(* Logix 5000 project; controller WWTP_SEC_CLX vendor 1 type 14 code 54 rev 17.2; software revision 17.00; part 11 of 13 *)

VAR_GLOBAL   (* controller tags *)
   BLR400_Fault : P_DIn := (Inp_Gate := 1, Cfg_NormTextVis := 1, Cfg_PCmdClear := 1, Cfg_HasTgtDisagreeAlm := 1, Cfg_TgtDisagreeAckReqd := 1, Cfg_TgtDisagreeSeverity := 3, Cfg_TgtDisagreeMinDuration := 5, Sts_SubstPV := 1, Ack_TgtDisagree := 1, Rdy_InpPV := 1);   // Secondary Treatment BLR-400 Fault
   BLR400_Intlk : P_Intlk := (Cfg_Latched := 2#0000_0000_0000_0001, Cfg_Bypassable := 2#0000_0000_0000_0001, Cfg_PCmdClear := 1, Sts_NBIntlkOK := 1, Sts_Intlk := 2#0000_0000_0000_0001, Sts_FirstOut := 2#0000_0000_0000_0001, Rdy_Reset := 1);   // BLR-400 Interlock
   BLR400_Motor : P_Motor := (Inp_PermOK := 1, Inp_NBPermOK := 1, Inp_NBIntlkOK := 1, Cfg_HasRunFdbk := 1, Cfg_UseRunFdbk := 1, Cfg_HasPermObj := 1, Cfg_HasIntlkObj := 1, Cfg_HasResInhObj := 1, Cfg_HasRunTimeObj := 1, Cfg_HasFailToStartAlm := 1, Cfg_HasFailToStopAlm := 1, Cfg_HasIntlkTripAlm := 1, Cfg_FailToStartAckReqd := 1, Cfg_FailToStopAckReqd := 1, Cfg_IntlkTripAckReqd := 1, Cfg_IOFaultAckReqd := 1, Cfg_FailToStartSeverity := 4, Cfg_FailToStopSeverity := 4, Cfg_IntlkTripSeverity := 2, Cfg_IOFaultSeverity := 4, Cfg_SimFdbkT := 2, Cfg_FailToStartT := 10, Cfg_FailToStopT := 10, PCmd_Start := 1, PCmd_Acq := 1, Sts_Stopped := 1, Sts_Oper := 1, Sts_ProgOperLock := 1, Ack_FailToStart := 1, Ack_FailToStop := 1, Ack_IntlkTrip := 1, Ack_IOFault := 1, Rdy_Bypass := 1, Rdy_Disable := 1);   // BLR-400 Motor
   BLR400_Perm : P_Perm := (Inp_Perm00 := 1, Inp_Perm01 := 1, Inp_Perm02 := 1, Inp_Perm03 := 1, Inp_Perm04 := 1, Inp_Perm05 := 1, Inp_Perm06 := 1, Inp_Perm07 := 1, Inp_Perm08 := 1, Inp_Perm09 := 1, Inp_Perm10 := 1, Inp_Perm11 := 1, Inp_Perm12 := 1, Inp_Perm13 := 1, Inp_Perm14 := 1, Inp_Perm15 := 1, Cfg_Bypassable := 2#0000_0000_0000_0001, Sts_PermOK := 1, Sts_NBPermOK := 1, Sts_Perm := 2#1111_1111_1111_1111);   // BLR-400 Permissive
   BLR400_Reset : P_Reset := (Inp_ResetReqd := 1, Cfg_MinHoldTime := 1, Rdy_Reset := 1);   // BLR-400 Reset
   BLR400_ResInh : P_ResInh := (Inp_Stopped := 1, Cfg_ThreeColdStarts := 1800, Cfg_FirstFailCold := 1800, Cfg_SubseqFailCold := 14400, Cfg_FirstFailHot := 1800, Cfg_SubseqFailHot := 14400, Cfg_HotRestartOK := 3600, Cfg_RestartHot := 3600, Cfg_HotToCold := 57600, Val_State := 1, Sts_Ready := 1);   // BLR-400 Restart Inhibit
   BLR400_RunTime : P_RunTime := (Cfg_PCmdClear := 1, Val_Starts := 14, Val_CurRunHrs := 0.0007652778, Val_MaxRunHrs := 0.37565723, Val_TotRunHrs := 0.7);   // BLR-400 Run Time
   I_BLR400_Fault : ALIAS FOR Local:2:I.DATA.2;
   I_BLR400_Fault_IOFault : ALIAS FOR Local:2:I.Fault.2;
   I_BLR400_InAuto : ALIAS FOR Local:2:I.DATA.0;
   I_BLR400_InAuto_IOFault : ALIAS FOR Local:2:I.Fault.0;
   I_BLR400_RunFdbk : ALIAS FOR Local:2:I.DATA.1;
   I_BLR400_RunFdbk_IOFault : ALIAS FOR Local:2:I.Fault.1;
   I_M400_Fault : ALIAS FOR Local:2:I.DATA.10;
   I_M400_Fault_IOFault : ALIAS FOR Local:2:I.Fault.10;
   I_M400_InAuto : ALIAS FOR Local:2:I.DATA.11;
   I_M400_InAuto_IOFault : ALIAS FOR Local:2:I.Fault.11;
   I_M400_RunFdbk : ALIAS FOR Local:2:I.DATA.9;
   I_M400_RunFdbk_IOFault : ALIAS FOR Local:2:I.Fault.9;
   I_M401_Fault : ALIAS FOR Local:2:I.DATA.13;
   I_M401_Fault_IOFault : ALIAS FOR Local:2:I.Fault.13;
   I_M401_InAuto : ALIAS FOR Local:2:I.DATA.14;
   I_M401_InAuto_IOFault : ALIAS FOR Local:2:I.Fault.14;
   I_M401_RunFdbk : ALIAS FOR Local:2:I.DATA.12;
   I_M401_RunFdbk_IOFault : ALIAS FOR Local:2:I.Fault.12;
   I_M402_Fault : ALIAS FOR Local:3:I.DATA.1;
   I_M402_Fault_IOFault : ALIAS FOR Local:3:I.Fault.1;
   I_M402_InAuto : ALIAS FOR Local:3:I.DATA.2;
   I_M402_InAuto_IOFault : ALIAS FOR Local:3:I.Fault.2;
   I_M402_RunFdbk : ALIAS FOR Local:3:I.DATA.0;
   I_M402_RunFdbk_IOFault : ALIAS FOR Local:3:I.Fault.0;
   I_M403_Fault : ALIAS FOR Local:3:I.DATA.4;
   I_M403_Fault_IOFault : ALIAS FOR Local:3:I.Fault.4;
   I_M403_InAuto : ALIAS FOR Local:3:I.DATA.5;
   I_M403_InAuto_IOFault : ALIAS FOR Local:3:I.Fault.5;
   I_M403_RunFdbk : ALIAS FOR Local:3:I.DATA.3;
   I_M403_RunFdbk_IOFault : ALIAS FOR Local:3:I.Fault.3;
   I_SecTk01_InAuto : ALIAS FOR Local:2:I.DATA.4;
   I_SecTk01_InAuto_IOFault : ALIAS FOR Local:2:I.Fault.4;
   I_SecTk01_RAS_Flow : ALIAS FOR Local:5:I.CH0DATA;
   I_SecTk01_RAS_Flow_IOFault : ALIAS FOR Local:5:I.CH0Fault;
   I_SecTk01_RunFdbk : ALIAS FOR Local:2:I.DATA.3;
   I_SecTk01_RunFdbk_IOFault : ALIAS FOR Local:2:I.Fault.3;
   I_SecTk01_Torque : ALIAS FOR Local:2:I.DATA.5;
   I_SecTk01_Torque_IOFault : ALIAS FOR Local:2:I.Fault.5;
   I_SecTk02_InAuto : ALIAS FOR Local:2:I.DATA.7;
   I_SecTk02_InAuto_IOFault : ALIAS FOR Local:2:I.Fault.7;
   I_SecTk02_RAS_Flow : ALIAS FOR Local:5:I.CH1DATA;
   I_SecTk02_RAS_Flow_IOFault : ALIAS FOR Local:5:I.CH1Fault;
   I_SecTk02_RunFdbk : ALIAS FOR Local:2:I.DATA.6;
   I_SecTk02_RunFdbk_IOFault : ALIAS FOR Local:2:I.Fault.6;
   I_SecTk02_Torque : ALIAS FOR Local:2:I.DATA.8;
   I_SecTk02_Torque_IOFault : ALIAS FOR Local:2:I.Fault.8;
   M400_Fault : P_DIn := (Inp_Gate := 1, Cfg_NormTextVis := 1, Cfg_PCmdClear := 1, Cfg_TgtDisagreeAckReqd := 1, Cfg_TgtDisagreeSeverity := 3, Sts_InpPV := 1, Ack_TgtDisagree := 1, Rdy_SubstPV := 1);   // Secondary Treatment M-400 Fault
   M400_Intlk : P_Intlk := (Cfg_PCmdClear := 1, Sts_IntlkOK := 1, Sts_NBIntlkOK := 1);   // M-400 Interlock
   M400_Motor : P_Motor := (Inp_PermOK := 1, Inp_NBPermOK := 1, Inp_IntlkOK := 1, Inp_NBIntlkOK := 1, Inp_IOFault := 1, Cfg_FailToStartAckReqd := 1, Cfg_FailToStopAckReqd := 1, Cfg_IntlkTripAckReqd := 1, Cfg_IOFaultAckReqd := 1, Cfg_FailToStartSeverity := 4, Cfg_FailToStopSeverity := 4, Cfg_IntlkTripSeverity := 2, Cfg_IOFaultSeverity := 4, Cfg_SimFdbkT := 2, Cfg_FailToStartT := 10, Cfg_FailToStopT := 10, PCmd_Acq := 1, Out_Stop := 1, Sts_Stopped := 1, Sts_Prog := 1, Ack_FailToStart := 1, Ack_FailToStop := 1, Ack_IntlkTrip := 1, Sts_IOFault := 1, Ack_IOFault := 1, Rdy_Bypass := 1, Rdy_Disable := 1);   // M-400 Motor
   M400_Perm : P_Perm := (Inp_Perm00 := 1, Inp_Perm01 := 1, Inp_Perm02 := 1, Inp_Perm03 := 1, Inp_Perm04 := 1, Inp_Perm05 := 1, Inp_Perm06 := 1, Inp_Perm07 := 1, Inp_Perm08 := 1, Inp_Perm09 := 1, Inp_Perm10 := 1, Inp_Perm11 := 1, Inp_Perm12 := 1, Inp_Perm13 := 1, Inp_Perm14 := 1, Inp_Perm15 := 1, Sts_PermOK := 1, Sts_NBPermOK := 1, Sts_Perm := 2#1111_1111_1111_1111);   // M-400 Permissive
   M400_Reset : P_Reset := (Cfg_MinHoldTime := 1);   // M-400 Reset
   M400_ResInh : P_ResInh := (Inp_Stopped := 1, Cfg_ThreeColdStarts := 1800, Cfg_FirstFailCold := 1800, Cfg_SubseqFailCold := 14400, Cfg_FirstFailHot := 1800, Cfg_SubseqFailHot := 14400, Cfg_HotRestartOK := 3600, Cfg_RestartHot := 3600, Cfg_HotToCold := 57600, Val_State := 1, Sts_Ready := 1);   // M-400 Restart Inhibit
   M400_RunTime : P_RunTime := (Cfg_PCmdClear := 1);   // M-400 Run Time
   M401_Fault : P_DIn := (Inp_PVBad := 1, Inp_Gate := 1, Cfg_NormTextVis := 1, Cfg_PCmdClear := 1, Cfg_TgtDisagreeAckReqd := 1, Cfg_TgtDisagreeSeverity := 3, Sts_InpPV := 1, Sts_PVBad := 1, Ack_TgtDisagree := 1, Rdy_SubstPV := 1);   // Secondary Treatment M-401 Fault
   M401_Fault_01 : P_DIn := (Inp_PV := 1, Inp_Target := 1, Inp_Gate := 1, Cfg_NormTextVis := 1, Cfg_PCmdClear := 1, Cfg_TgtDisagreeAckReqd := 1, Cfg_TgtDisagreeSeverity := 3);
   M401_Intlk : P_Intlk := (Cfg_PCmdClear := 1, Sts_IntlkOK := 1, Sts_NBIntlkOK := 1);   // M-401 Interlock
   M401_Intlk_01 : P_Intlk := (Cfg_PCmdClear := 1, Sts_IntlkOK := 1, Sts_NBIntlkOK := 1);
   M401_Motor : P_Motor := (Inp_PermOK := 1, Inp_NBPermOK := 1, Inp_IntlkOK := 1, Inp_NBIntlkOK := 1, Inp_IOFault := 1, Cfg_FailToStartAckReqd := 1, Cfg_FailToStopAckReqd := 1, Cfg_IntlkTripAckReqd := 1, Cfg_IOFaultAckReqd := 1, Cfg_FailToStartSeverity := 4, Cfg_FailToStopSeverity := 4, Cfg_IntlkTripSeverity := 2, Cfg_IOFaultSeverity := 4, Cfg_SimFdbkT := 2, Cfg_FailToStartT := 10, Cfg_FailToStopT := 10, PCmd_Acq := 1, Out_Stop := 1, Sts_Stopped := 1, Sts_Prog := 1, Ack_FailToStart := 1, Ack_FailToStop := 1, Ack_IntlkTrip := 1, Sts_IOFault := 1, Ack_IOFault := 1, Rdy_Bypass := 1, Rdy_Disable := 1);   // M-401 Motor
   M401_Motor_01 : P_Motor := (Inp_PermOK := 1, Inp_NBPermOK := 1, Inp_IntlkOK := 1, Inp_NBIntlkOK := 1, Cfg_PCmdClear := 1, Cfg_FailToStartAckReqd := 1, Cfg_FailToStopAckReqd := 1, Cfg_IntlkTripAckReqd := 1, Cfg_IOFaultAckReqd := 1, Cfg_FailToStartSeverity := 4, Cfg_FailToStopSeverity := 4, Cfg_IntlkTripSeverity := 2, Cfg_IOFaultSeverity := 4, Cfg_SimFdbkT := 2, Cfg_FailToStartT := 10, Cfg_FailToStopT := 10, Sts_Stopped := 1, Sts_Oper := 1);
   M401_Perm : P_Perm := (Inp_Perm00 := 1, Inp_Perm01 := 1, Inp_Perm02 := 1, Inp_Perm03 := 1, Inp_Perm04 := 1, Inp_Perm05 := 1, Inp_Perm06 := 1, Inp_Perm07 := 1, Inp_Perm08 := 1, Inp_Perm09 := 1, Inp_Perm10 := 1, Inp_Perm11 := 1, Inp_Perm12 := 1, Inp_Perm13 := 1, Inp_Perm14 := 1, Inp_Perm15 := 1, Sts_PermOK := 1, Sts_NBPermOK := 1, Sts_Perm := 2#1111_1111_1111_1111);   // M-401 Permissive
   M401_Perm_01 : P_Perm := (Inp_Perm00 := 1, Inp_Perm01 := 1, Inp_Perm02 := 1, Inp_Perm03 := 1, Inp_Perm04 := 1, Inp_Perm05 := 1, Inp_Perm06 := 1, Inp_Perm07 := 1, Inp_Perm08 := 1, Inp_Perm09 := 1, Inp_Perm10 := 1, Inp_Perm11 := 1, Inp_Perm12 := 1, Inp_Perm13 := 1, Inp_Perm14 := 1, Inp_Perm15 := 1, Sts_PermOK := 1, Sts_NBPermOK := 1, Sts_Perm := 2#1111_1111_1111_1111);
   M401_Reset : P_Reset := (Cfg_MinHoldTime := 1);   // M-401 Reset
   M401_Reset_01 : P_Reset := (Inp_ResetReqd := 1, Cfg_MinHoldTime := 1, Rdy_Reset := 1);
   M401_ResInh : P_ResInh := (Inp_Stopped := 1, Cfg_ThreeColdStarts := 1800, Cfg_FirstFailCold := 1800, Cfg_SubseqFailCold := 14400, Cfg_FirstFailHot := 1800, Cfg_SubseqFailHot := 14400, Cfg_HotRestartOK := 3600, Cfg_RestartHot := 3600, Cfg_HotToCold := 57600, Val_State := 1, Sts_Ready := 1);   // M-401 Restart Inhibit
   M401_ResInh_01 : P_ResInh := (Inp_Running := 1, Cfg_ThreeColdStarts := 1800, Cfg_FirstFailCold := 1800, Cfg_SubseqFailCold := 14400, Cfg_FirstFailHot := 1800, Cfg_SubseqFailHot := 14400, Cfg_HotRestartOK := 3600, Cfg_RestartHot := 3600, Cfg_HotToCold := 57600, Val_State := 1);
   M401_RunTime : P_RunTime := (Cfg_PCmdClear := 1);   // M-401 Run Time
   M401_RunTime_01 : P_RunTime := (Inp_Running := 1, Cfg_PCmdClear := 1);
   M402_Fault : P_DIn := (Inp_PVBad := 1, Inp_Gate := 1, Cfg_NormTextVis := 1, Cfg_PCmdClear := 1, Cfg_TgtDisagreeAckReqd := 1, Cfg_TgtDisagreeSeverity := 3, Sts_InpPV := 1, Sts_PVBad := 1, Ack_TgtDisagree := 1, Rdy_SubstPV := 1);   // Secondary Treatment M-402 Fault
   M402_Fault_01 : P_DIn := (Inp_PV := 1, Inp_Target := 1, Inp_Gate := 1, Cfg_NormTextVis := 1, Cfg_PCmdClear := 1, Cfg_TgtDisagreeAckReqd := 1, Cfg_TgtDisagreeSeverity := 3);
   M402_Intlk : P_Intlk := (Cfg_PCmdClear := 1, Sts_IntlkOK := 1, Sts_NBIntlkOK := 1);   // M-402 Interlock
   M402_Intlk_01 : P_Intlk := (Cfg_PCmdClear := 1, Sts_IntlkOK := 1, Sts_NBIntlkOK := 1);
   M402_Motor : P_Motor := (Inp_PermOK := 1, Inp_NBPermOK := 1, Inp_IntlkOK := 1, Inp_NBIntlkOK := 1, Inp_IOFault := 1, Cfg_FailToStartAckReqd := 1, Cfg_FailToStopAckReqd := 1, Cfg_IntlkTripAckReqd := 1, Cfg_IOFaultAckReqd := 1, Cfg_FailToStartSeverity := 4, Cfg_FailToStopSeverity := 4, Cfg_IntlkTripSeverity := 2, Cfg_IOFaultSeverity := 4, Cfg_SimFdbkT := 2, Cfg_FailToStartT := 10, Cfg_FailToStopT := 10, PCmd_Acq := 1, Out_Stop := 1, Sts_Stopped := 1, Sts_Prog := 1, Ack_FailToStart := 1, Ack_FailToStop := 1, Ack_IntlkTrip := 1, Sts_IOFault := 1, Ack_IOFault := 1, Rdy_Bypass := 1, Rdy_Disable := 1);   // M-402 Motor
   M402_Motor_01 : P_Motor := (Inp_PermOK := 1, Inp_NBPermOK := 1, Inp_IntlkOK := 1, Inp_NBIntlkOK := 1, Cfg_PCmdClear := 1, Cfg_FailToStartAckReqd := 1, Cfg_FailToStopAckReqd := 1, Cfg_IntlkTripAckReqd := 1, Cfg_IOFaultAckReqd := 1, Cfg_FailToStartSeverity := 4, Cfg_FailToStopSeverity := 4, Cfg_IntlkTripSeverity := 2, Cfg_IOFaultSeverity := 4, Cfg_SimFdbkT := 2, Cfg_FailToStartT := 10, Cfg_FailToStopT := 10, Sts_Stopped := 1, Sts_Oper := 1);
   M402_Perm : P_Perm := (Inp_Perm00 := 1, Inp_Perm01 := 1, Inp_Perm02 := 1, Inp_Perm03 := 1, Inp_Perm04 := 1, Inp_Perm05 := 1, Inp_Perm06 := 1, Inp_Perm07 := 1, Inp_Perm08 := 1, Inp_Perm09 := 1, Inp_Perm10 := 1, Inp_Perm11 := 1, Inp_Perm12 := 1, Inp_Perm13 := 1, Inp_Perm14 := 1, Inp_Perm15 := 1, Sts_PermOK := 1, Sts_NBPermOK := 1, Sts_Perm := 2#1111_1111_1111_1111);   // M-402 Permissive
   M402_Perm_01 : P_Perm := (Inp_Perm00 := 1, Inp_Perm01 := 1, Inp_Perm02 := 1, Inp_Perm03 := 1, Inp_Perm04 := 1, Inp_Perm05 := 1, Inp_Perm06 := 1, Inp_Perm07 := 1, Inp_Perm08 := 1, Inp_Perm09 := 1, Inp_Perm10 := 1, Inp_Perm11 := 1, Inp_Perm12 := 1, Inp_Perm13 := 1, Inp_Perm14 := 1, Inp_Perm15 := 1, Sts_PermOK := 1, Sts_NBPermOK := 1, Sts_Perm := 2#1111_1111_1111_1111);
   M402_Reset : P_Reset := (Cfg_MinHoldTime := 1);   // M-402 Reset
   M402_Reset_01 : P_Reset := (Inp_ResetReqd := 1, Cfg_MinHoldTime := 1, Rdy_Reset := 1);
   M402_ResInh : P_ResInh := (Inp_Stopped := 1, Cfg_ThreeColdStarts := 1800, Cfg_FirstFailCold := 1800, Cfg_SubseqFailCold := 14400, Cfg_FirstFailHot := 1800, Cfg_SubseqFailHot := 14400, Cfg_HotRestartOK := 3600, Cfg_RestartHot := 3600, Cfg_HotToCold := 57600, Val_State := 1, Sts_Ready := 1);   // M-402 Restart Inhibit
   M402_ResInh_01 : P_ResInh := (Inp_Running := 1, Cfg_ThreeColdStarts := 1800, Cfg_FirstFailCold := 1800, Cfg_SubseqFailCold := 14400, Cfg_FirstFailHot := 1800, Cfg_SubseqFailHot := 14400, Cfg_HotRestartOK := 3600, Cfg_RestartHot := 3600, Cfg_HotToCold := 57600, Val_State := 1);
   M402_RunTime : P_RunTime := (Cfg_PCmdClear := 1);   // M-402 Run Time
   M402_RunTime_01 : P_RunTime := (Inp_Running := 1, Cfg_PCmdClear := 1);
   M403_Fault : P_DIn := (Inp_PVBad := 1, Inp_Gate := 1, Cfg_NormTextVis := 1, Cfg_PCmdClear := 1, Cfg_TgtDisagreeAckReqd := 1, Cfg_TgtDisagreeSeverity := 3, Sts_InpPV := 1, Sts_PVBad := 1, Ack_TgtDisagree := 1, Rdy_SubstPV := 1);   // Secondary Treatment M-403 Fault
   M403_Intlk : P_Intlk := (Cfg_PCmdClear := 1, Sts_IntlkOK := 1, Sts_NBIntlkOK := 1);   // M-403 Interlock
   M403_Motor : P_Motor := (Inp_PermOK := 1, Inp_NBPermOK := 1, Inp_IntlkOK := 1, Inp_NBIntlkOK := 1, Inp_IOFault := 1, Cfg_FailToStartAckReqd := 1, Cfg_FailToStopAckReqd := 1, Cfg_IntlkTripAckReqd := 1, Cfg_IOFaultAckReqd := 1, Cfg_FailToStartSeverity := 4, Cfg_FailToStopSeverity := 4, Cfg_IntlkTripSeverity := 2, Cfg_IOFaultSeverity := 4, Cfg_SimFdbkT := 2, Cfg_FailToStartT := 10, Cfg_FailToStopT := 10, PCmd_Acq := 1, Out_Stop := 1, Sts_Stopped := 1, Sts_Prog := 1, Ack_FailToStart := 1, Ack_FailToStop := 1, Ack_IntlkTrip := 1, Sts_IOFault := 1, Ack_IOFault := 1, Rdy_Bypass := 1, Rdy_Disable := 1);   // M-403 Motor
   M403_Perm : P_Perm := (Inp_Perm00 := 1, Inp_Perm01 := 1, Inp_Perm02 := 1, Inp_Perm03 := 1, Inp_Perm04 := 1, Inp_Perm05 := 1, Inp_Perm06 := 1, Inp_Perm07 := 1, Inp_Perm08 := 1, Inp_Perm09 := 1, Inp_Perm10 := 1, Inp_Perm11 := 1, Inp_Perm12 := 1, Inp_Perm13 := 1, Inp_Perm14 := 1, Inp_Perm15 := 1, Sts_PermOK := 1, Sts_NBPermOK := 1, Sts_Perm := 2#1111_1111_1111_1111);   // M-403 Permissive
   M403_Reset : P_Reset := (Cfg_MinHoldTime := 1);   // M-403 Reset
   M403_ResInh : P_ResInh := (Inp_Stopped := 1, Cfg_ThreeColdStarts := 1800, Cfg_FirstFailCold := 1800, Cfg_SubseqFailCold := 14400, Cfg_FirstFailHot := 1800, Cfg_SubseqFailHot := 14400, Cfg_HotRestartOK := 3600, Cfg_RestartHot := 3600, Cfg_HotToCold := 57600, Val_State := 1, Sts_Ready := 1);   // M-403 Restart Inhibit
   M403_RunTime : P_RunTime := (Cfg_PCmdClear := 1);   // M-403 Run Time
   O_BLR400_Out_Run : ALIAS FOR Local:4:O.DATA.2;   // BLR-400 Start/Stop
   O_M400_Out_Run : ALIAS FOR Local:4:O.DATA.3;   // M-400 Start/Stop
   O_M401_Out_Run : ALIAS FOR Local:4:O.DATA.4;   // M-401 Start/Stop
   O_M402_Out_Run : ALIAS FOR Local:4:O.DATA.5;   // M-402 Start/Stop
   O_M403_Out_Run : ALIAS FOR Local:4:O.DATA.6;   // M-402 Start/Stop
   O_SecTk01_Out_Run : ALIAS FOR Local:4:O.DATA.0;   // Secondary Tank #1 Start/Stop
   O_SecTk02_Out_Run : ALIAS FOR Local:4:O.DATA.1;   // Secondary Tank #2 Start/Stop
   PLC_CommFail : U_CommFail := (Inp_Heartbeat := 1, CFG_DelayTimerSec := 30, Sts_CommFail := 1);
   PLC_Device_ResetPB : BOOL;   // Site Wide Device Reset Push Button
   PLC_Heartbeat : U_Heartbeat := (CFG_DelayTimerSec := 30, Heartbeat := 1);   // PLC Heartbeat
   PLC_Simulation : BOOL;   // Application running IN SIMULATION
   PLC_WallClock : U_WallClock := (Val_CurrentYear := 1998, Val_CurrentMonth := 2, Val_CurrentDay := 24, Val_CurrentMinute := 29, Val_CurrentSecond := 56, Val_DayOfWeek := 2);   // Wall Clock
   PRIM_FLOW_FIT302 : P_AIn := (Cfg_SetTrack := 1, Cfg_PCmdClear := 1, Cfg_HiHiAckReqd := 1, Cfg_HiAckReqd := 1, Cfg_LoAckReqd := 1, Cfg_LoLoAckReqd := 1, Cfg_FailAckReqd := 1, Cfg_HiHiSeverity := 3, Cfg_HiSeverity := 2, Cfg_LoSeverity := 2, Cfg_LoLoSeverity := 3, Cfg_FailSeverity := 4, Cfg_InpRawMax := 100.0, Cfg_PVEUMax := 100.0, Cfg_HiHiDB := 1.0, Cfg_HiDB := 1.0, Cfg_LoDB := 1.0, Cfg_LoLoDB := 1.0, Cfg_FailHiLim := 1.5e+38, Cfg_FailLoLim := -1.5e+38, PSet_HiHiLim := 1.5e+38, PSet_HiLim := 1.5e+38, PSet_LoLim := -1.5e+38, PSet_LoLoLim := -1.5e+38, OSet_HiHiLim := 1.5e+38, OSet_HiLim := 1.5e+38, OSet_LoLim := -1.5e+38, OSet_LoLoLim := -1.5e+38, Val_PVEUMax := 100.0, Val_HiHiLim := 1.5e+38, Val_HiLim := 1.5e+38, Val_LoLim := -1.5e+38, Val_LoLoLim := -1.5e+38, Sts_InpPV := 1, Sts_Oper := 1);   // Primary Treatment Flow (FIT-302)
   RAS_P401_DischFlow_AIn : P_AIn := (Inp_PV := 3.0, Cfg_SetTrack := 1, Cfg_PCmdClear := 1, Cfg_HiHiAckReqd := 1, Cfg_HiAckReqd := 1, Cfg_LoAckReqd := 1, Cfg_LoLoAckReqd := 1, Cfg_FailAckReqd := 1, Cfg_HiHiSeverity := 3, Cfg_HiSeverity := 2, Cfg_LoSeverity := 2, Cfg_LoLoSeverity := 3, Cfg_FailSeverity := 4, Cfg_InpRawMax := 3.0, Cfg_PVEUMax := 3.0, Cfg_HiHiDB := 1.0, Cfg_HiDB := 1.0, Cfg_LoDB := 1.0, Cfg_LoLoDB := 1.0, Cfg_FailHiLim := 21.0, Cfg_FailLoLim := -1.0, PSet_HiHiLim := 1.5e+38, PSet_HiLim := 1.5e+38, PSet_LoLim := -1.5e+38, PSet_LoLoLim := -1.5e+38, MSet_SubstPV := 3.0, OSet_HiHiLim := 1.5e+38, OSet_HiLim := 1.5e+38, OSet_LoLim := -1.5e+38, OSet_LoLoLim := -1.5e+38, Set_SimPV := 3.0, Val := 3.0, Val_InpPV := 3.0, Val_PVEUMax := 3.0, Val_HiHiLim := 1.5e+38, Val_HiLim := 1.5e+38, Val_LoLim := -1.5e+38, Val_LoLoLim := -1.5e+38, Sts_InpPV := 1, Sts_Oper := 1, Ack_HiHi := 1, Ack_Hi := 1, Ack_Lo := 1, Ack_LoLo := 1, Ack_Fail := 1);   // Secondary Treament Tank #1 RAS Flow (FIT-400)
   RAS_P401_DischFlow_Tot : U_FlowTot := (Inp_ProgStartReq := 1, Val_FlowRate := 3.0, Val_DailyTot := 6236.7607, Val_YestTot := 33286.41, Val_YearlyTot := 1.4820616);   // Secondary Treament Tank #1 RAS Flow (FIT-400) Totalizer
   RAS_P401_Intlk : P_Intlk := (Cfg_PCmdClear := 1, Sts_IntlkOK := 1, Sts_NBIntlkOK := 1);   // Secondary Treatment RAS Pump #401 Interlock
   RAS_P401_Perm : P_Perm := (Inp_Perm00 := 1, Inp_Perm01 := 1, Inp_Perm02 := 1, Inp_Perm03 := 1, Inp_Perm04 := 1, Inp_Perm05 := 1, Inp_Perm06 := 1, Inp_Perm07 := 1, Inp_Perm08 := 1, Inp_Perm09 := 1, Inp_Perm10 := 1, Inp_Perm11 := 1, Inp_Perm12 := 1, Inp_Perm13 := 1, Inp_Perm14 := 1, Inp_Perm15 := 1, Cfg_Bypassable := 2#0000_0000_0000_0001, Sts_PermOK := 1, Sts_NBPermOK := 1, Sts_Perm := 2#1111_1111_1111_1111);   // Secondary Treatment RAS Pump #401 Permissive
   RAS_P401_PIDE : PID_ENHANCED := (PV := 20.0, PVEUMax := 100.0, SPHLimit := 100.0, UseRatio := 1, RatioProg := 1.0, RatioOper := 1.0, RatioHLimit := 100.0, CVEUMax := 60.0, CVHLimit := 100.0, PGain := 1.0, PVEDerivative := 1, AllowCasRat := 1, ProgAutoReq := 1, RTSTime := 1, CVLAlarm := 1, PVPercent := 20.0, E := -20.0, EPercent := -20.0, WindupLOut := 1, Ratio := 1.0, CasRat := 1, DeltaT := 0.007);   // Secondary Treatment RAS Pump #401 PIDE
   RAS_P401_PIDE_AutoTune : PIDE_AUTOTUNE;   // Secondary Treatment RAS Pump #401 PIDE AutoTune
   RAS_P401_Reset : P_Reset := (Cfg_MinHoldTime := 1);   // Secondary Treatment RAS Pump #401 Reset
   RAS_P401_ResInh : P_ResInh := (Inp_Stopped := 1, Cfg_ThreeColdStarts := 1800, Cfg_FirstFailCold := 1800, Cfg_SubseqFailCold := 14400, Cfg_FirstFailHot := 1800, Cfg_SubseqFailHot := 14400, Cfg_HotRestartOK := 3600, Cfg_RestartHot := 60, Cfg_HotToCold := 57600, Val_State := 1, Sts_Ready := 1);   // Secondary Treatment RAS Pump #401 Restart Inhibit
   RAS_P401_RunTime : P_RunTime := (Cfg_PCmdClear := 1, Val_Starts := 44, Val_CurRunHrs := 0.105334446, Val_MaxRunHrs := 22.180851, Val_TotRunHrs := 26.2);   // Secondary Treatment RAS Pump #401 Run Time
   RAS_P401_VSD : P_VSD := (Inp_FaultCode := 75, Inp_Datalink := 200, Inp_Ready := 1, Inp_CommandDir := 1, Inp_ActualDir := 1, Inp_FwdPermOK := 1, Inp_FwdNBPermOK := 1, Inp_RevPermOK := 1, Inp_RevNBPermOK := 1, Inp_IntlkOK := 1, Inp_NBIntlkOK := 1, Cfg_HasRunFdbk := 1, Cfg_UseRunFdbk := 1, Cfg_HasInpDatalink := 1, Cfg_HasOutDatalink := 1, Cfg_HasFwdPermObj := 1, Cfg_HasIntlkObj := 1, Cfg_HasResInhObj := 1, Cfg_HasRunTimeObj := 1, Cfg_SetTrack := 1, Cfg_HasFailToStartAlm := 1, Cfg_HasFailToStopAlm := 1, Cfg_HasDriveFaultAlm := 1, Cfg_FailToStartAckReqd := 1, Cfg_FailToStopAckReqd := 1, Cfg_IntlkTripAckReqd := 1, Cfg_DriveFaultAckReqd := 1, Cfg_IOFaultAckReqd := 1, Cfg_FailToStartSeverity := 4, Cfg_FailToStopSeverity := 4, Cfg_IntlkTripSeverity := 2, Cfg_DriveFaultSeverity := 4, Cfg_IOFaultSeverity := 4, Cfg_MaxSpdRef := 60.0, Cfg_SpeedRefRawMax := 32767, Cfg_SpeedRefEUMax := 130.0, Cfg_SpeedFdbkRawMax := 32767, Cfg_SpeedFdbkEUMax := 130.0, Cfg_InpDatalinkRawMax := 4095, Cfg_InpDatalinkEUMax := 409.5, Cfg_OutDatalinkMax := 100.0, Cfg_OutDatalinkRawMax := 4095, Cfg_OutDatalinkEUMax := 409.5, Cfg_SimRampT := 10, Cfg_FailToStartT := 15, Cfg_FailToStopT := 15, Cfg_ResetPulseT := 2, PSet_SpeedRef := 20.0, OSet_SpeedRef := 20.0, OSet_OutDatalink := 20.0, PCmd_Acq := 1, Out_SpeedRef := 5041, Out_Datalink := 200, Out_Fwd := 1, Val_SpeedRef := 20.0, Val_InpDatalink := 20.0, Val_OutDatalink := 20.0, Val_SpeedFdbkEUMax := 130.0, Sts_Stopped := 1, Sts_CommandDir := 1,
        Sts_ActualDir := 1, Sts_Oper := 1, Sts_ProgOperLock := 1, Ack_FailToStart := 1, Ack_FailToStop := 1, Ack_IntlkTrip := 1, Ack_DriveFault := 1, Ack_IOFault := 1, Rdy_Start := 1, Rdy_Bypass := 1, Rdy_Disable := 1);   // Secondary Treatment RAS Pump #401 Variable Speed Drive
   RAS_P402_DischFlow_Tot : U_FlowTot := (Inp_ProgStartReq := 1, Val_FlowRate := 20.0, Val_DailyTot := 108682.97, Val_YearlyTot := 1.0868297);   // Secondary Treament Tank #2 RAS Flow (FIT-401) Totalizer
   RAS_P402_Intlk : P_Intlk := (Cfg_PCmdClear := 1, Sts_IntlkOK := 1, Sts_NBIntlkOK := 1);   // Secondary Treatment RAS Pump #402 Interlock
   RAS_P402_Perm : P_Perm := (Inp_Perm01 := 1, Inp_Perm02 := 1, Inp_Perm03 := 1, Inp_Perm04 := 1, Inp_Perm05 := 1, Inp_Perm06 := 1, Inp_Perm07 := 1, Inp_Perm08 := 1, Inp_Perm09 := 1, Inp_Perm10 := 1, Inp_Perm11 := 1, Inp_Perm12 := 1, Inp_Perm13 := 1, Inp_Perm14 := 1, Inp_Perm15 := 1, Sts_Perm := 2#1111_1111_1111_1110);   // Secondary Treatment RAS Pump #402 Permissive
   RAS_P402_Reset : P_Reset := (Cfg_MinHoldTime := 1);   // Secondary Treatment RAS Pump #402 Reset
   RAS_P402_ResInh : P_ResInh := (Inp_Running := 1, Cfg_ThreeColdStarts := 1800, Cfg_FirstFailCold := 1800, Cfg_SubseqFailCold := 14400, Cfg_FirstFailHot := 1800, Cfg_SubseqFailHot := 14400, Cfg_HotRestartOK := 3600, Cfg_RestartHot := 3600, Cfg_HotToCold := 57600, Val_MinToReady := 4, Val_SecToReady := 9, Val_State := 8);   // Secondary Treatment RAS Pump #402 Restart Inhibit
   RAS_P402_RunTime : P_RunTime := (Inp_Running := 1, Cfg_PCmdClear := 1, Val_Starts := 33, Val_CurRunHrs := 0.06839083, Val_MaxRunHrs := 0.06839083, Val_TotRunHrs := 0.2);   // Secondary Treatment RAS Pump #402 Run Time
   RAS_P402_VSD : P_VSD := (Inp_Ready := 1, Inp_CommandDir := 1, Inp_ActualDir := 1, Inp_FwdPermOK := 1, Inp_FwdNBPermOK := 1, Inp_RevPermOK := 1, Inp_RevNBPermOK := 1, Inp_IntlkOK := 1, Inp_NBIntlkOK := 1, Cfg_HasRunFdbk := 1, Cfg_UseRunFdbk := 1, Cfg_SetTrack := 1, Cfg_PCmdClear := 1, Cfg_DriveFaultResetReqd := 1, Cfg_FailToStartAckReqd := 1, Cfg_FailToStopAckReqd := 1, Cfg_IntlkTripAckReqd := 1, Cfg_IOFaultAckReqd := 1, Cfg_FailToStartSeverity := 4, Cfg_FailToStopSeverity := 4, Cfg_IntlkTripSeverity := 2, Cfg_DriveFaultSeverity := 4, Cfg_IOFaultSeverity := 4, Cfg_MaxSpdRef := 60.0, Cfg_SpeedRefRawMax := 32767, Cfg_SpeedRefEUMax := 130.0, Cfg_SpeedFdbkRawMax := 32767, Cfg_SpeedFdbkEUMax := 130.0, Cfg_InpDatalinkRawMax := 4095, Cfg_InpDatalinkEUMax := 409.5, Cfg_OutDatalinkMax := 100.0, Cfg_OutDatalinkRawMax := 4095, Cfg_OutDatalinkEUMax := 409.5, Cfg_SimRampT := 10, Cfg_FailToStartT := 15, Cfg_FailToStopT := 15, Cfg_ResetPulseT := 2, Val_SpeedFdbkEUMax := 130.0, Sts_Stopped := 1, Sts_CommandDir := 1, Sts_ActualDir := 1, Sts_Oper := 1);   // Secondary Treatment RAS Pump #402 VSD
   RAS_P403_DischFlow_AIn : P_AIn := (Inp_PV := 20.0, Cfg_SetTrack := 1, Cfg_PCmdClear := 1, Cfg_HiHiAckReqd := 1, Cfg_HiAckReqd := 1, Cfg_LoAckReqd := 1, Cfg_LoLoAckReqd := 1, Cfg_FailAckReqd := 1, Cfg_HiHiSeverity := 3, Cfg_HiSeverity := 2, Cfg_LoSeverity := 2, Cfg_LoLoSeverity := 3, Cfg_FailSeverity := 4, Cfg_InpRawMax := 20.0, Cfg_PVEUMax := 20.0, Cfg_HiHiDB := 1.0, Cfg_HiDB := 1.0, Cfg_LoDB := 1.0, Cfg_LoLoDB := 1.0, Cfg_FailHiLim := 21.0, Cfg_FailLoLim := -1.0, PSet_HiHiLim := 1.5e+38, PSet_HiLim := 1.5e+38, PSet_LoLim := -1.5e+38, PSet_LoLoLim := -1.5e+38, MSet_SubstPV := 20.0, OSet_HiHiLim := 1.5e+38, OSet_HiLim := 1.5e+38, OSet_LoLim := -1.5e+38, OSet_LoLoLim := -1.5e+38, Set_SimPV := 20.0, Val := 20.0, Val_InpPV := 20.0, Val_PVEUMax := 20.0, Val_HiHiLim := 1.5e+38, Val_HiLim := 1.5e+38, Val_LoLim := -1.5e+38, Val_LoLoLim := -1.5e+38, Sts_InpPV := 1, Sts_Oper := 1, Sts_ProgOperLock := 1, Ack_HiHi := 1, Ack_Hi := 1, Ack_Lo := 1, Ack_LoLo := 1, Ack_Fail := 1);   // Secondary Treament Tank #2 RAS Flow (FIT-401)
   SecTk01_Intlk : P_Intlk := (Cfg_Latched := 2#0000_0000_0000_0001, Cfg_Bypassable := 2#0000_0000_0000_0001, Cfg_PCmdClear := 1, Sts_NBIntlkOK := 1, Sts_Intlk := 2#0000_0000_0000_0001, Sts_FirstOut := 2#0000_0000_0000_0001, Rdy_Reset := 1);   // Secondary Treatment Tank #1 Interlock
   SecTk01_Motor : P_Motor := (Inp_PermOK := 1, Inp_NBPermOK := 1, Inp_NBIntlkOK := 1, Cfg_HasRunFdbk := 1, Cfg_UseRunFdbk := 1, Cfg_HasPermObj := 1, Cfg_HasIntlkObj := 1, Cfg_HasResInhObj := 1, Cfg_HasRunTimeObj := 1, Cfg_HasFailToStartAlm := 1, Cfg_HasFailToStopAlm := 1, Cfg_HasIntlkTripAlm := 1, Cfg_FailToStartAckReqd := 1, Cfg_FailToStopAckReqd := 1, Cfg_IntlkTripAckReqd := 1, Cfg_IOFaultAckReqd := 1, Cfg_FailToStartSeverity := 4, Cfg_FailToStopSeverity := 4, Cfg_IntlkTripSeverity := 4, Cfg_IOFaultSeverity := 4, Cfg_SimFdbkT := 2, Cfg_FailToStartT := 10, Cfg_FailToStopT := 10, PCmd_Start := 1, PCmd_Acq := 1, Sts_Stopped := 1, Sts_Oper := 1, Sts_ProgOperLock := 1, Ack_FailToStart := 1, Ack_FailToStop := 1, Ack_IntlkTrip := 1, Ack_IOFault := 1, Rdy_Bypass := 1, Rdy_Disable := 1);   // Secondary Treatment Tank #1 Motor
   SecTk01_Perm : P_Perm := (Inp_Perm00 := 1, Inp_Perm01 := 1, Inp_Perm02 := 1, Inp_Perm03 := 1, Inp_Perm04 := 1, Inp_Perm05 := 1, Inp_Perm06 := 1, Inp_Perm07 := 1, Inp_Perm08 := 1, Inp_Perm09 := 1, Inp_Perm10 := 1, Inp_Perm11 := 1, Inp_Perm12 := 1, Inp_Perm13 := 1, Inp_Perm14 := 1, Inp_Perm15 := 1, Cfg_Bypassable := 2#0000_0000_0000_0001, Sts_PermOK := 1, Sts_NBPermOK := 1, Sts_Perm := 2#1111_1111_1111_1111);   // Secondary Treatment Tank #1 Permissive
   SecTk01_Reset : P_Reset := (Inp_ResetReqd := 1, Cfg_MinHoldTime := 1, Rdy_Reset := 1);   // Secondary Treatment Tank #1 Reset
   SecTk01_ResInh : P_ResInh := (Inp_Stopped := 1, Cfg_ThreeColdStarts := 1800, Cfg_FirstFailCold := 1800, Cfg_SubseqFailCold := 14400, Cfg_FirstFailHot := 1800, Cfg_SubseqFailHot := 14400, Cfg_HotRestartOK := 3600, Cfg_RestartHot := 3600, Cfg_HotToCold := 57600, Val_State := 1, Sts_Ready := 1);   // Secondary Treatment Tank #1 Restart Inhibit
   SecTk01_RunTime : P_RunTime := (Cfg_PCmdClear := 1, Val_Starts := 36, Val_CurRunHrs := 0.0038158332, Val_MaxRunHrs := 4.4467525, Val_TotRunHrs := 4.7000003);   // Secondary Treatment Tank #1 Run Time
   SecTk01_Torque : P_DIn := (Inp_PV := 1, Inp_Gate := 1, Cfg_NormTextVis := 1, Cfg_PCmdClear := 1, Cfg_HasTgtDisagreeAlm := 1, Cfg_TgtDisagreeAckReqd := 1, Cfg_TgtDisagreeSeverity := 3, Cfg_TgtDisagreeMinDuration := 5, Set_SimPV := 1, Sts_PV := 1, Sts_SubstPV := 1, Ack_TgtDisagree := 1, Rdy_InpPV := 1);   // Secondary Treatment Tank #1 Torque Fault
   SecTk02_Intlk : P_Intlk := (Cfg_PCmdClear := 1, Sts_IntlkOK := 1, Sts_NBIntlkOK := 1);   // Secondary Treatment Tank #2 Interlock
   SecTk02_Motor : P_Motor := (Inp_PermOK := 1, Inp_NBPermOK := 1, Inp_IntlkOK := 1, Inp_NBIntlkOK := 1, Cfg_HasRunFdbk := 1, Cfg_UseRunFdbk := 1, Cfg_HasPermObj := 1, Cfg_HasIntlkObj := 1, Cfg_HasResInhObj := 1, Cfg_HasRunTimeObj := 1, Cfg_HasFailToStartAlm := 1, Cfg_HasFailToStopAlm := 1, Cfg_FailToStartAckReqd := 1, Cfg_FailToStopAckReqd := 1, Cfg_IntlkTripAckReqd := 1, Cfg_IOFaultAckReqd := 1, Cfg_FailToStartSeverity := 4, Cfg_FailToStopSeverity := 4, Cfg_IntlkTripSeverity := 2, Cfg_IOFaultSeverity := 4, Cfg_SimFdbkT := 2, Cfg_FailToStartT := 10, Cfg_FailToStopT := 10, PCmd_Stop := 1, PCmd_Acq := 1, Val_Notify := 1, Sts_Stopped := 1, Sts_Available := 1, Sts_Prog := 1, Ack_FailToStart := 1, Ack_IntlkTrip := 1, Ack_IOFault := 1, Rdy_Bypass := 1, Rdy_Disable := 1);   // Secondary Treatment Tank #2 Motor
   SecTk02_Perm : P_Perm := (Inp_Perm00 := 1, Inp_Perm01 := 1, Inp_Perm02 := 1, Inp_Perm03 := 1, Inp_Perm04 := 1, Inp_Perm05 := 1, Inp_Perm06 := 1, Inp_Perm07 := 1, Inp_Perm08 := 1, Inp_Perm09 := 1, Inp_Perm10 := 1, Inp_Perm11 := 1, Inp_Perm12 := 1, Inp_Perm13 := 1, Inp_Perm14 := 1, Inp_Perm15 := 1, Sts_PermOK := 1, Sts_NBPermOK := 1, Sts_Perm := 2#1111_1111_1111_1111);   // Secondary Treatment Tank #2 Permissive
   SecTk02_Reset : P_Reset := (Cfg_MinHoldTime := 1);   // Secondary Treatment Tank #2 Reset
   SecTk02_ResInh : P_ResInh := (Inp_Stopped := 1, Cfg_ThreeColdStarts := 1800, Cfg_FirstFailCold := 1800, Cfg_SubseqFailCold := 14400, Cfg_FirstFailHot := 1800, Cfg_SubseqFailHot := 14400, Cfg_HotRestartOK := 3600, Cfg_RestartHot := 3600, Cfg_HotToCold := 57600, Val_State := 1, Sts_Ready := 1);   // Secondary Treatment Tank #2 Restart Inhibit
   SecTk02_RunTime : P_RunTime := (Cfg_PCmdClear := 1, Val_Starts := 16, Val_CurRunHrs := 0.01666611, Val_MaxRunHrs := 0.01666611);   // Secondary Treatment Tank #2 Run Time
   SecTk02_Torque : P_DIn := (Inp_Gate := 1, Cfg_NormTextVis := 1, Cfg_PCmdClear := 1, Cfg_TgtDisagreeAckReqd := 1, Cfg_TgtDisagreeSeverity := 3, Sts_InpPV := 1, Ack_TgtDisagree := 1, Rdy_SubstPV := 1);   // Secondary Treatment Tank #2 Torque Fault
   WTP_P401_VFD_Input : AB:PowerFlex700AC_Drive_Parameters:I:0;
   WTP_P401_VFD_Output : AB:PowerFlex700AC_Drive_Parameters:O:0;
END_VAR

PROGRAM AerationBlower   (* main routine Main *)
VAR
   Equip_Fault : ALIAS FOR I_BLR400_Fault;
   Equip_Fault_IOFault : ALIAS FOR I_BLR400_Fault_IOFault;
   Equip_GroupReset : ALIAS FOR PLC_Device_ResetPB;
   Equip_InAuto : ALIAS FOR I_BLR400_InAuto;
   Equip_InAuto_IOFault : ALIAS FOR I_BLR400_InAuto_IOFault;
   Equip_Intlk : ALIAS FOR BLR400_Intlk;
   Equip_IOFault : BOOL;
   Equip_Motor : ALIAS FOR BLR400_Motor;
   Equip_Out_Run : ALIAS FOR O_BLR400_Out_Run;
   Equip_RunFdbk : ALIAS FOR I_BLR400_RunFdbk;
   Equip_RunFdbk_IOFault : ALIAS FOR I_BLR400_RunFdbk_IOFault;
   Wrk_Hand : BOOL;
   Wrk_ResetReqd : BOOL := 1;
   Wrk_ResetRequired : BOOL;
END_VAR

ROUTINE A01_Blower_LDR   (* ladder *)
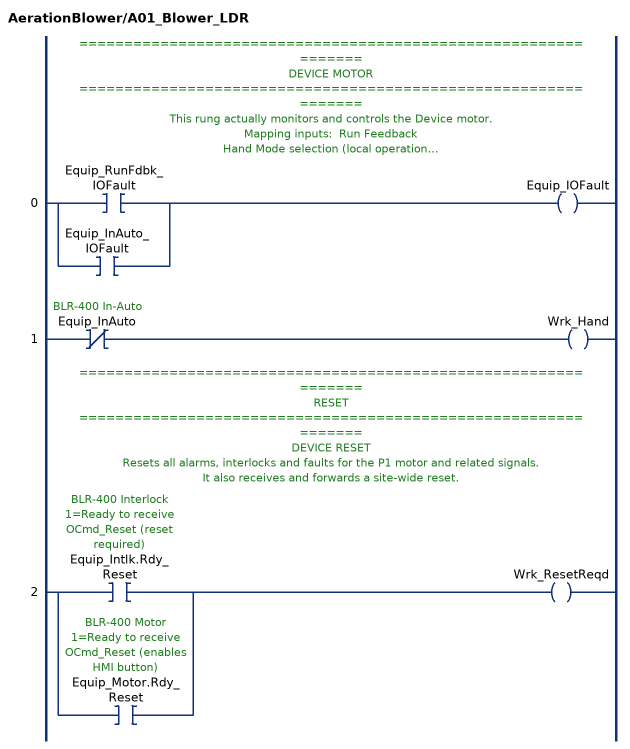
   // ===============================================================
   // DEVICE MOTOR
   // ===============================================================
   // This rung actually monitors and controls the Device motor.
   // Mapping inputs:  Run Feedback
   // Hand Mode selection (local operation)
   // Permissive OK
   // Protective’s OK,
   // I/O Fault signals
   // Pump Reset (above)
   // DEVICE
   // Output Mapping: Starter output
   0: [XIC(Equip_RunFdbk_IOFault) ,XIC(Equip_InAuto_IOFault) ]OTE(Equip_IOFault);
   1: XIO(Equip_InAuto)OTE(Wrk_Hand);
   // ===============================================================
   // RESET
   // ===============================================================
   // DEVICE RESET
   // Resets all alarms, interlocks and faults for the P1 motor and related signals.
   // It also receives and forwards a site-wide reset.
   2: [XIC(Equip_Intlk.Rdy_Reset) ,XIC(Equip_Motor.Rdy_Reset) ]OTE(Wrk_ResetReqd);
END_ROUTINE

ROUTINE A02_Blower_FBD   (* function block diagram *)
   SHEET 1   // Motor
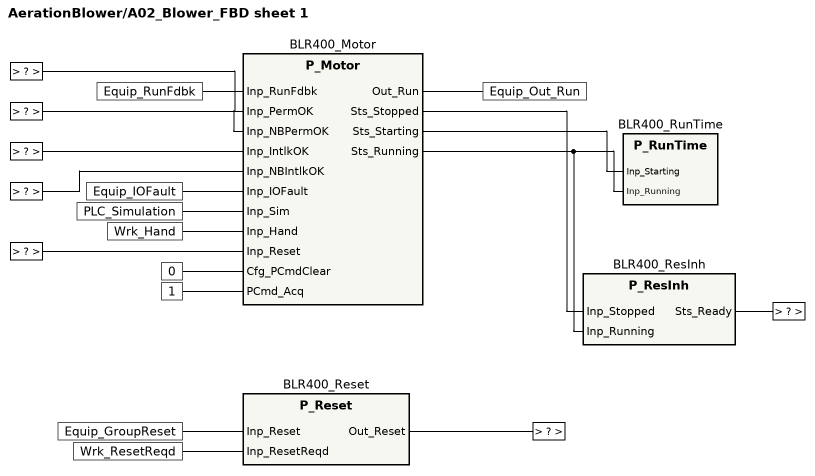
   BLR400_Reset : P_Reset(Inp_Reset := Equip_GroupReset, Inp_ResetReqd := Wrk_ResetReqd);
   WIRE(?) := BLR400_Reset.Out_Reset;
   BLR400_ResInh : P_ResInh(Inp_Stopped := BLR400_Motor.Sts_Stopped {feedback}, Inp_Running := BLR400_Motor.Sts_Running {feedback});
   WIRE(?) := BLR400_ResInh.Sts_Ready;
   BLR400_Motor : P_Motor(Inp_RunFdbk := Equip_RunFdbk, Inp_PermOK := WIRE(?), Inp_NBPermOK := WIRE(?), Inp_IntlkOK := WIRE(?), Inp_NBIntlkOK := WIRE(?), Inp_IOFault := Equip_IOFault, Inp_Sim := PLC_Simulation, Inp_Hand := Wrk_Hand, Inp_Reset := WIRE(?), Cfg_PCmdClear := 0, PCmd_Acq := 1);
   Equip_Out_Run := BLR400_Motor.Out_Run;
   BLR400_RunTime : P_RunTime(Inp_Starting := BLR400_Motor.Sts_Starting, Inp_Running := BLR400_Motor.Sts_Running);
   SHEET 2   // Permissives / Interlocks
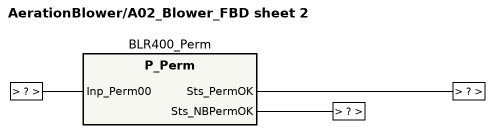
   BLR400_Perm : P_Perm(Inp_Perm00 := WIRE(?));
   WIRE(?) := BLR400_Perm.Sts_NBPermOK;
   WIRE(?) := BLR400_Perm.Sts_PermOK;
   SHEET 3   // Interlocks
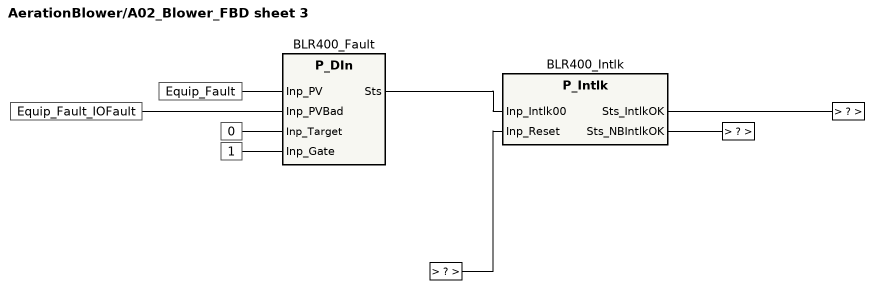
   BLR400_Fault : P_DIn(Inp_PV := Equip_Fault, Inp_PVBad := Equip_Fault_IOFault, Inp_Target := 0, Inp_Gate := 1);
   BLR400_Intlk : P_Intlk(Inp_Intlk00 := BLR400_Fault.Sts, Inp_Reset := WIRE(?));
   WIRE(?) := BLR400_Intlk.Sts_NBIntlkOK;
   WIRE(?) := BLR400_Intlk.Sts_IntlkOK;
END_ROUTINE

ROUTINE Main   (* ladder *)
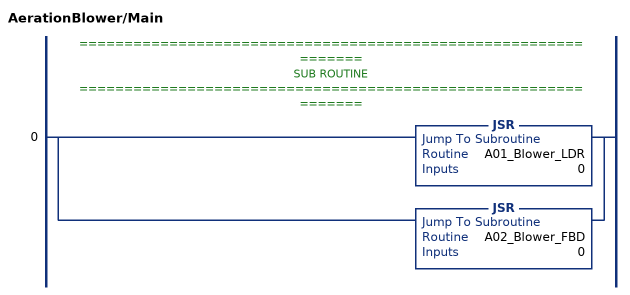
   // ===============================================================
   // SUB ROUTINE
   // ===============================================================
   0: [JSR(A01_Blower_LDR,0) ,JSR(A02_Blower_FBD,0) ];
END_ROUTINE
END_PROGRAM

PROGRAM AerationTk01_Mixer01   (* main routine Main *)
VAR
   Equip_Fault : ALIAS FOR I_M400_Fault;
   Equip_Fault_IOFault : ALIAS FOR I_M400_Fault_IOFault;
   Equip_GroupReset : ALIAS FOR PLC_Device_ResetPB;
   Equip_InAuto : ALIAS FOR I_M400_InAuto;
   Equip_InAuto_IOFault : ALIAS FOR I_M400_InAuto_IOFault;
   Equip_Intlk : ALIAS FOR M400_Intlk;
   Equip_IOFault : BOOL := 1;
   Equip_Motor : ALIAS FOR M400_Motor;
   Equip_Out_Run : ALIAS FOR O_M400_Out_Run;
   Equip_RunFdbk : ALIAS FOR I_M400_RunFdbk;
   Equip_RunFdbk_IOFault : ALIAS FOR I_M400_RunFdbk_IOFault;
   Wrk_Hand : BOOL;
   Wrk_ResetReqd : BOOL;
   Wrk_ResetRequired : BOOL;
END_VAR

ROUTINE A01_Mixer_LDR   (* ladder *)
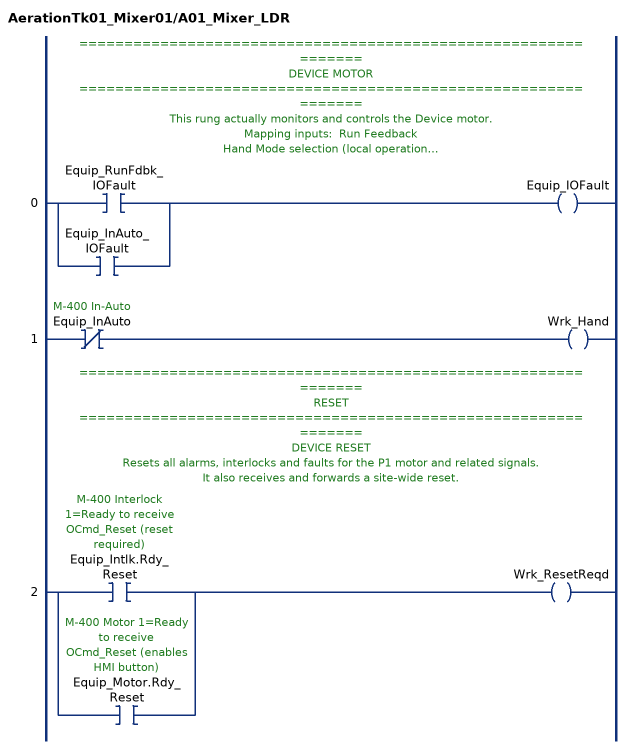
   // ===============================================================
   // DEVICE MOTOR
   // ===============================================================
   // This rung actually monitors and controls the Device motor.
   // Mapping inputs:  Run Feedback
   // Hand Mode selection (local operation)
   // Permissive OK
   // Protective’s OK,
   // I/O Fault signals
   // Pump Reset (above)
   // DEVICE
   // Output Mapping: Starter output
   0: [XIC(Equip_RunFdbk_IOFault) ,XIC(Equip_InAuto_IOFault) ]OTE(Equip_IOFault);
   1: XIO(Equip_InAuto)OTE(Wrk_Hand);
   // ===============================================================
   // RESET
   // ===============================================================
   // DEVICE RESET
   // Resets all alarms, interlocks and faults for the P1 motor and related signals.
   // It also receives and forwards a site-wide reset.
   2: [XIC(Equip_Intlk.Rdy_Reset) ,XIC(Equip_Motor.Rdy_Reset) ]OTE(Wrk_ResetReqd);
END_ROUTINE

ROUTINE A02_Mixer_FBD   (* function block diagram *)
   SHEET 1   // Motor
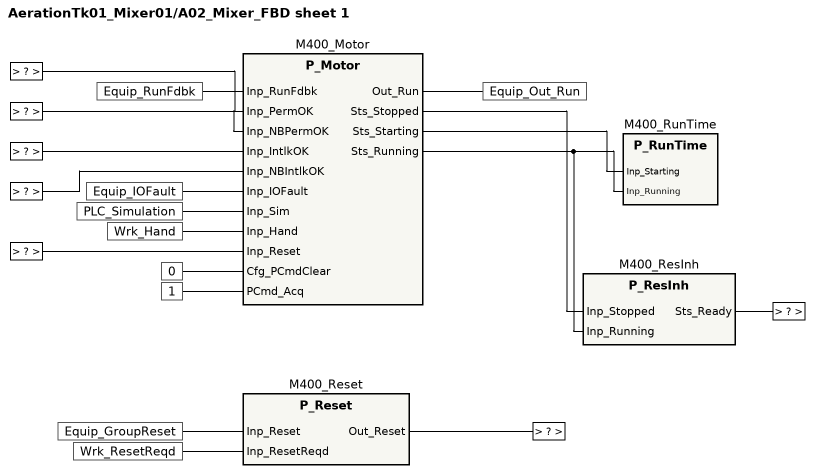
   M400_Reset : P_Reset(Inp_Reset := Equip_GroupReset, Inp_ResetReqd := Wrk_ResetReqd);
   WIRE(?) := M400_Reset.Out_Reset;
   M400_ResInh : P_ResInh(Inp_Stopped := M400_Motor.Sts_Stopped {feedback}, Inp_Running := M400_Motor.Sts_Running {feedback});
   WIRE(?) := M400_ResInh.Sts_Ready;
   M400_Motor : P_Motor(Inp_RunFdbk := Equip_RunFdbk, Inp_PermOK := WIRE(?), Inp_NBPermOK := WIRE(?), Inp_IntlkOK := WIRE(?), Inp_NBIntlkOK := WIRE(?), Inp_IOFault := Equip_IOFault, Inp_Sim := PLC_Simulation, Inp_Hand := Wrk_Hand, Inp_Reset := WIRE(?), Cfg_PCmdClear := 0, PCmd_Acq := 1);
   Equip_Out_Run := M400_Motor.Out_Run;
   M400_RunTime : P_RunTime(Inp_Starting := M400_Motor.Sts_Starting, Inp_Running := M400_Motor.Sts_Running);
   SHEET 2   // Permissives / Interlocks
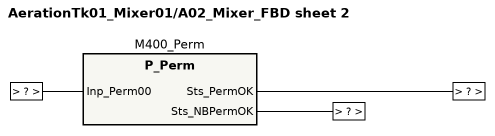
   M400_Perm : P_Perm(Inp_Perm00 := WIRE(?));
   WIRE(?) := M400_Perm.Sts_NBPermOK;
   WIRE(?) := M400_Perm.Sts_PermOK;
   SHEET 3   // Interlocks
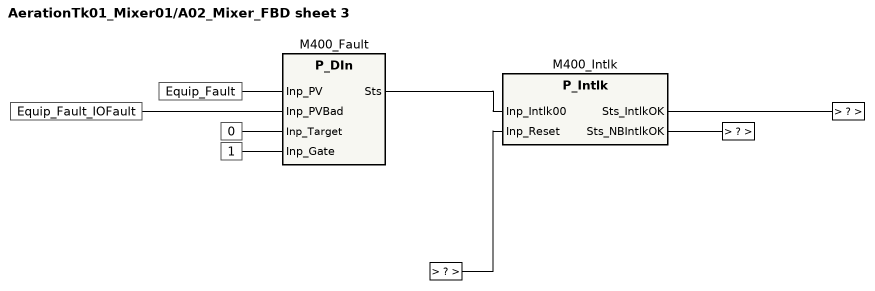
   M400_Fault : P_DIn(Inp_PV := Equip_Fault, Inp_PVBad := Equip_Fault_IOFault, Inp_Target := 0, Inp_Gate := 1);
   M400_Intlk : P_Intlk(Inp_Intlk00 := M400_Fault.Sts, Inp_Reset := WIRE(?));
   WIRE(?) := M400_Intlk.Sts_NBIntlkOK;
   WIRE(?) := M400_Intlk.Sts_IntlkOK;
END_ROUTINE

ROUTINE Main   (* ladder *)
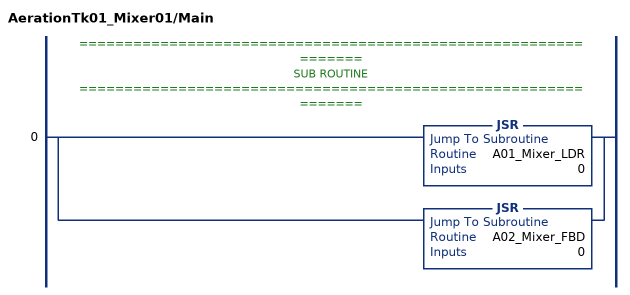
   // ===============================================================
   // SUB ROUTINE
   // ===============================================================
   0: [JSR(A01_Mixer_LDR,0) ,JSR(A02_Mixer_FBD,0) ];
END_ROUTINE
END_PROGRAM

PROGRAM AerationTk01_Mixer02   (* main routine Main *)
VAR
   Equip_Fault : ALIAS FOR I_M401_Fault;
   Equip_Fault_IOFault : ALIAS FOR I_M401_Fault_IOFault;
   Equip_GroupReset : ALIAS FOR PLC_Device_ResetPB;
   Equip_InAuto : ALIAS FOR I_M401_InAuto;
   Equip_InAuto_IOFault : ALIAS FOR I_M401_InAuto_IOFault;
   Equip_Intlk : ALIAS FOR M401_Intlk;
   Equip_IOFault : BOOL := 1;
   Equip_Motor : ALIAS FOR M401_Motor;
   Equip_Out_Run : ALIAS FOR O_M401_Out_Run;
   Equip_RunFdbk : ALIAS FOR I_M401_RunFdbk;
   Equip_RunFdbk_IOFault : ALIAS FOR I_M401_RunFdbk_IOFault;
   Wrk_Hand : BOOL;
   Wrk_ResetReqd : BOOL;
   Wrk_ResetRequired : BOOL;
END_VAR

ROUTINE A01_Mixer_LDR   (* ladder *)
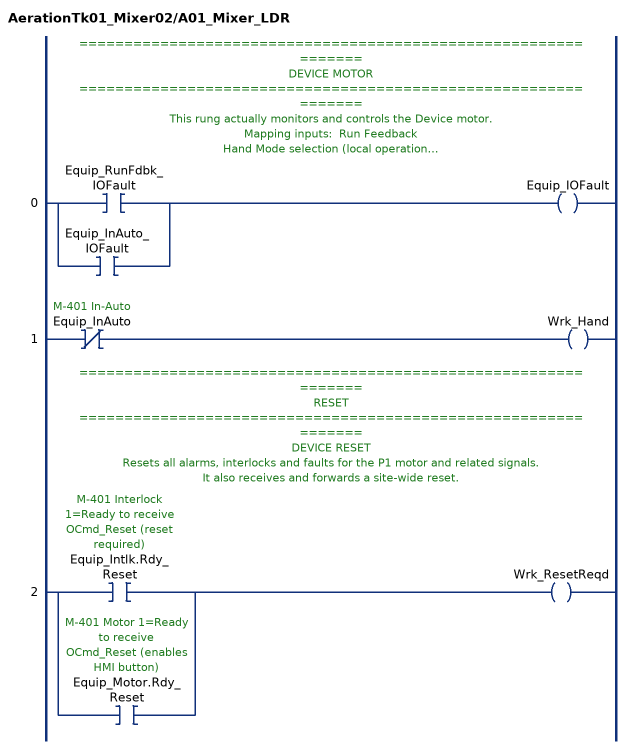
   // ===============================================================
   // DEVICE MOTOR
   // ===============================================================
   // This rung actually monitors and controls the Device motor.
   // Mapping inputs:  Run Feedback
   // Hand Mode selection (local operation)
   // Permissive OK
   // Protective’s OK,
   // I/O Fault signals
   // Pump Reset (above)
   // DEVICE
   // Output Mapping: Starter output
   0: [XIC(Equip_RunFdbk_IOFault) ,XIC(Equip_InAuto_IOFault) ]OTE(Equip_IOFault);
   1: XIO(Equip_InAuto)OTE(Wrk_Hand);
   // ===============================================================
   // RESET
   // ===============================================================
   // DEVICE RESET
   // Resets all alarms, interlocks and faults for the P1 motor and related signals.
   // It also receives and forwards a site-wide reset.
   2: [XIC(Equip_Intlk.Rdy_Reset) ,XIC(Equip_Motor.Rdy_Reset) ]OTE(Wrk_ResetReqd);
END_ROUTINE

ROUTINE A02_Mixer_FBD   (* function block diagram *)
   SHEET 1   // Motor
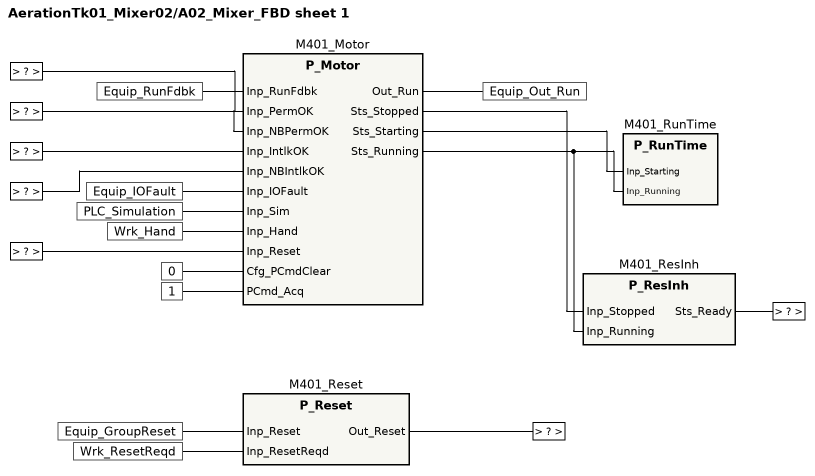
   M401_Reset : P_Reset(Inp_Reset := Equip_GroupReset, Inp_ResetReqd := Wrk_ResetReqd);
   WIRE(?) := M401_Reset.Out_Reset;
   M401_ResInh : P_ResInh(Inp_Stopped := M401_Motor.Sts_Stopped {feedback}, Inp_Running := M401_Motor.Sts_Running {feedback});
   WIRE(?) := M401_ResInh.Sts_Ready;
   M401_Motor : P_Motor(Inp_RunFdbk := Equip_RunFdbk, Inp_PermOK := WIRE(?), Inp_NBPermOK := WIRE(?), Inp_IntlkOK := WIRE(?), Inp_NBIntlkOK := WIRE(?), Inp_IOFault := Equip_IOFault, Inp_Sim := PLC_Simulation, Inp_Hand := Wrk_Hand, Inp_Reset := WIRE(?), Cfg_PCmdClear := 0, PCmd_Acq := 1);
   Equip_Out_Run := M401_Motor.Out_Run;
   M401_RunTime : P_RunTime(Inp_Starting := M401_Motor.Sts_Starting, Inp_Running := M401_Motor.Sts_Running);
   SHEET 2   // Permissives / Interlocks
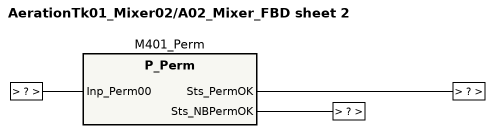
   M401_Perm : P_Perm(Inp_Perm00 := WIRE(?));
   WIRE(?) := M401_Perm.Sts_NBPermOK;
   WIRE(?) := M401_Perm.Sts_PermOK;
   SHEET 3   // Interlocks
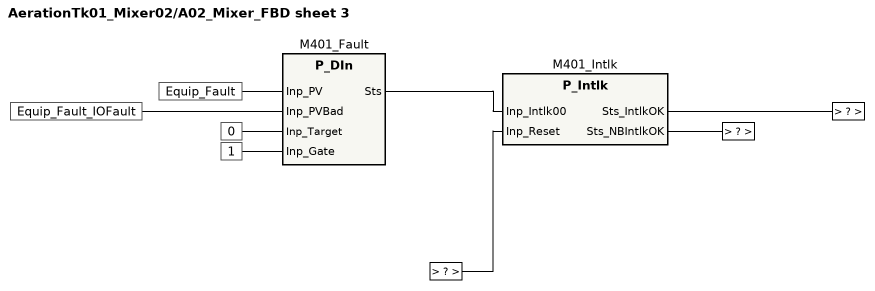
   M401_Fault : P_DIn(Inp_PV := Equip_Fault, Inp_PVBad := Equip_Fault_IOFault, Inp_Target := 0, Inp_Gate := 1);
   M401_Intlk : P_Intlk(Inp_Intlk00 := M401_Fault.Sts, Inp_Reset := WIRE(?));
   WIRE(?) := M401_Intlk.Sts_NBIntlkOK;
   WIRE(?) := M401_Intlk.Sts_IntlkOK;
END_ROUTINE

ROUTINE Main   (* ladder *)
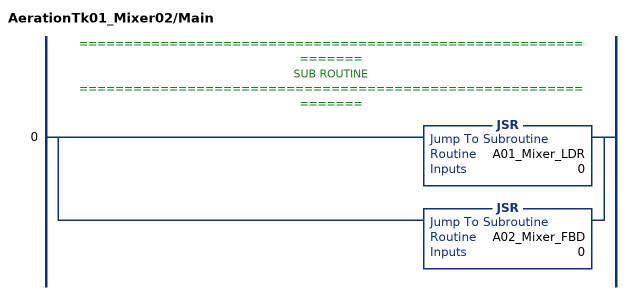
   // ===============================================================
   // SUB ROUTINE
   // ===============================================================
   0: [JSR(A01_Mixer_LDR,0) ,JSR(A02_Mixer_FBD,0) ];
END_ROUTINE
END_PROGRAM

PROGRAM AerationTk02_Mixer01   (* main routine Main *)
VAR
   Equip_Fault : ALIAS FOR I_M402_Fault;
   Equip_Fault_IOFault : ALIAS FOR I_M402_Fault_IOFault;
   Equip_GroupReset : ALIAS FOR PLC_Device_ResetPB;
   Equip_InAuto : ALIAS FOR I_M402_InAuto;
   Equip_InAuto_IOFault : ALIAS FOR I_M402_InAuto_IOFault;
   Equip_Intlk : ALIAS FOR M402_Intlk;
   Equip_IOFault : BOOL := 1;
   Equip_Motor : ALIAS FOR M402_Motor;
   Equip_Out_Run : ALIAS FOR O_M402_Out_Run;
   Equip_RunFdbk : ALIAS FOR I_M402_RunFdbk;
   Equip_RunFdbk_IOFault : ALIAS FOR I_M402_RunFdbk_IOFault;
   Wrk_Hand : BOOL;
   Wrk_ResetReqd : BOOL;
   Wrk_ResetRequired : BOOL;
END_VAR

ROUTINE A01_Mixer_LDR   (* ladder *)
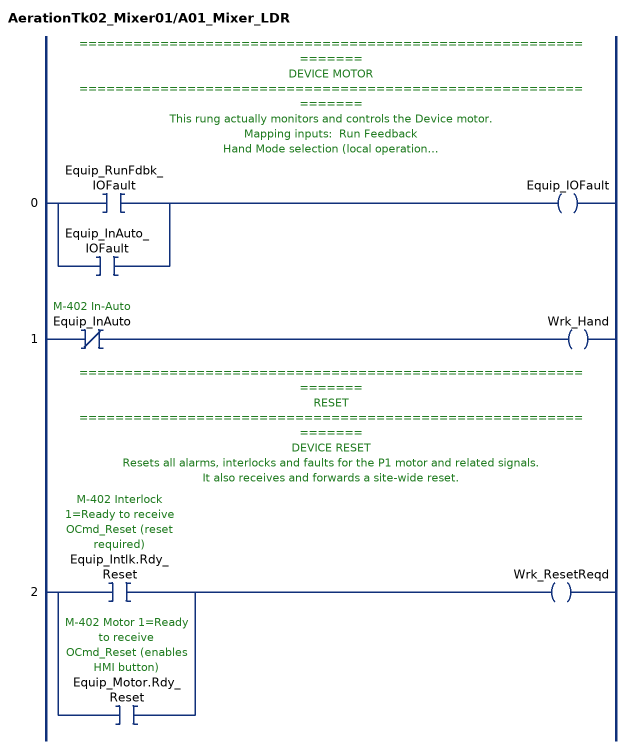
   // ===============================================================
   // DEVICE MOTOR
   // ===============================================================
   // This rung actually monitors and controls the Device motor.
   // Mapping inputs:  Run Feedback
   // Hand Mode selection (local operation)
   // Permissive OK
   // Protective’s OK,
   // I/O Fault signals
   // Pump Reset (above)
   // DEVICE
   // Output Mapping: Starter output
   0: [XIC(Equip_RunFdbk_IOFault) ,XIC(Equip_InAuto_IOFault) ]OTE(Equip_IOFault);
   1: XIO(Equip_InAuto)OTE(Wrk_Hand);
   // ===============================================================
   // RESET
   // ===============================================================
   // DEVICE RESET
   // Resets all alarms, interlocks and faults for the P1 motor and related signals.
   // It also receives and forwards a site-wide reset.
   2: [XIC(Equip_Intlk.Rdy_Reset) ,XIC(Equip_Motor.Rdy_Reset) ]OTE(Wrk_ResetReqd);
END_ROUTINE

ROUTINE A02_Mixer_FBD   (* function block diagram *)
   SHEET 1   // Motor
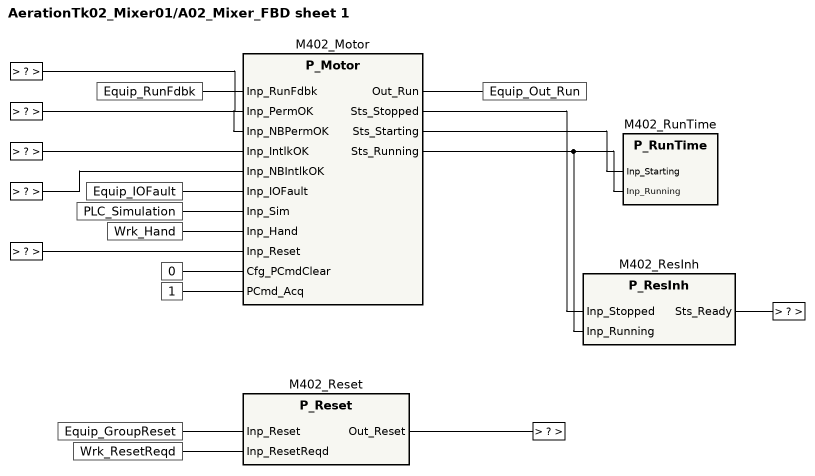
   M402_Reset : P_Reset(Inp_Reset := Equip_GroupReset, Inp_ResetReqd := Wrk_ResetReqd);
   WIRE(?) := M402_Reset.Out_Reset;
   M402_ResInh : P_ResInh(Inp_Stopped := M402_Motor.Sts_Stopped {feedback}, Inp_Running := M402_Motor.Sts_Running {feedback});
   WIRE(?) := M402_ResInh.Sts_Ready;
   M402_Motor : P_Motor(Inp_RunFdbk := Equip_RunFdbk, Inp_PermOK := WIRE(?), Inp_NBPermOK := WIRE(?), Inp_IntlkOK := WIRE(?), Inp_NBIntlkOK := WIRE(?), Inp_IOFault := Equip_IOFault, Inp_Sim := PLC_Simulation, Inp_Hand := Wrk_Hand, Inp_Reset := WIRE(?), Cfg_PCmdClear := 0, PCmd_Acq := 1);
   Equip_Out_Run := M402_Motor.Out_Run;
   M402_RunTime : P_RunTime(Inp_Starting := M402_Motor.Sts_Starting, Inp_Running := M402_Motor.Sts_Running);
   SHEET 2   // Permissives / Interlocks
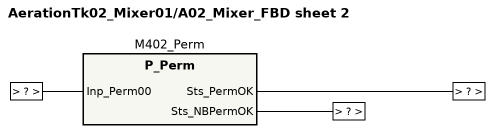
   M402_Perm : P_Perm(Inp_Perm00 := WIRE(?));
   WIRE(?) := M402_Perm.Sts_NBPermOK;
   WIRE(?) := M402_Perm.Sts_PermOK;
   SHEET 3   // Interlocks
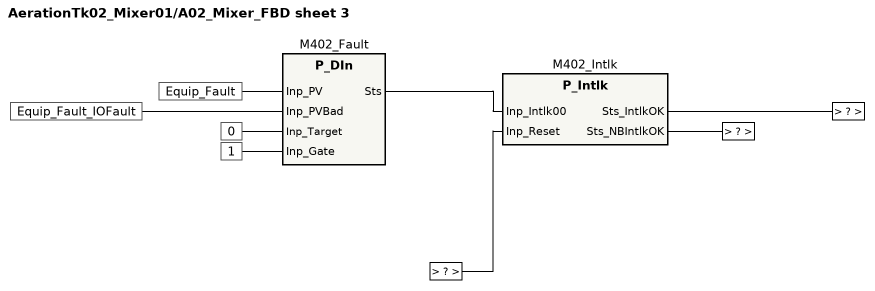
   M402_Fault : P_DIn(Inp_PV := Equip_Fault, Inp_PVBad := Equip_Fault_IOFault, Inp_Target := 0, Inp_Gate := 1);
   M402_Intlk : P_Intlk(Inp_Intlk00 := M402_Fault.Sts, Inp_Reset := WIRE(?));
   WIRE(?) := M402_Intlk.Sts_NBIntlkOK;
   WIRE(?) := M402_Intlk.Sts_IntlkOK;
END_ROUTINE
